Yaskawa INFORM job: 0_0.JBI

/JOB
//NAME 0_0
///FOLDERNAME OBROTNIK
//POS
///NPOS 0,0,1,0,0,0
///TOOL 0
///POSTYPE PULSE
///PULSE
EC00000=0,0
//INST
///DATE 2023/11/07 18:47
///ATTR SC,RW,RJ
////FRAME ROBOT
///GROUP1 ST1
NOP
MOVJ EC00000 VJ=100.00
END
